FUNCTION_BLOCK TreeStrategyExecutor EXTENDS CNM_AbstractObject.Object IMPLEMENTS CNM_CollectionInterfaces.ITreeStrategy
VAR
	tree :ITreeHelper;
	instantExecutor :InstantTreeStrategyExecutor;
END_VAR

(*

## Short summary

This abstract property returns the class name of the concrete object, 
which is useful for logging/debugging purpose.

.. <legal notes>

legal notes
=================
| SPDX-FileCopyrightText: © 2022 ekvip automation GmbH <info@ekvip.de>
| SPDX-License-Identifier: Apache-2.0
| For details check: Apache-2.0_

.. _Apache-2.0: https://www.apache.org/licenses/LICENSE-2.0

.. </legal notes>

*)
PROPERTY className : CNM_AbstractObject.ClassName
GET
className := 'CNM_Collections.TreeStrategyExecutor';
END_GET
END_PROPERTY

(*

## Short summary

The constructor ``FB_init`` is needed to create an unique hash code.
The hash code is a pseudo random number create with a [xorshift](https://en.wikipedia.org/wiki/Xorshift) algorithm.
It can be overwritten on derivations, because it will be called implicit, ``SUPER^.FB_init()`` is not required.
For more information check: [Behavoir with derived function blocks](https://infosys.beckhoff.com/content/1033/tc3_plc_intro/5482088715.html?id=6983869892358031022).

.. <legal notes>

legal notes
=================
| SPDX-FileCopyrightText: © 2022 ekvip automation GmbH <info@ekvip.de>
| SPDX-License-Identifier: Apache-2.0
| For details check: Apache-2.0_

.. _Apache-2.0: https://www.apache.org/licenses/LICENSE-2.0

.. </legal notes>


*)
METHOD FB_init : BOOL
VAR_INPUT
	(* if TRUE, the retain variables are initialized (warm start / cold start)*)
	bInitRetains	: BOOL;
	(* if TRUE, the instance afterwards gets moved into the copy code (online change) *)
	bInCopyCode	: BOOL;
	(*the tree which this executor will dispatch to*)
	tree :ITreeHelper;
END_VAR
THIS^.tree := tree;
THIS^.instantExecutor.assignTree(tree);
END_METHOD

(*

## Short summary

A method to insert a single element into the tree.

.. <legal notes>

legal notes
=================
| SPDX-FileCopyrightText: © 2022 ekvip automation GmbH <info@ekvip.de>
| SPDX-License-Identifier: Apache-2.0
| For details check: Apache-2.0_

.. _Apache-2.0: https://www.apache.org/licenses/LICENSE-2.0

.. </legal notes>


**Return:** ``SUCCESS``: operation successful
	``ABORTED``: operation was aborted (implementation specific)
	``ERROR``: out of memory

*)
METHOD insert : CNM_CollectionInterfaces.CNM_ReturnTypes.SingleExecutionResult
VAR_INPUT
	(*the object that should be inserted*)
	object	: CNM_CollectionInterfaces.CNM_AbstractObject.IObject;
END_VAR
insert := THIS^.tree.insert(object := object);
END_METHOD

(*

## Short summary

This method inserts all elements of a collection into the tree.

If any value of the collection could not be inserted because of duplication, operation isn't aborted, 
insertion is tried for every element of the collection.

.. <legal notes>

legal notes
=================
| SPDX-FileCopyrightText: © 2025 ekvip automation GmbH <info@ekvip.de>
| SPDX-License-Identifier: Apache-2.0
| For details check: Apache-2.0_

.. _Apache-2.0: https://www.apache.org/licenses/LICENSE-2.0

.. </legal notes>


**Return:** ``SUCCESS``: if insert could be made
	``ABORTED``: execute has a falling edge during insert,
	``BUSY``: Insert is in Progress
	``ERROR``: the passed collection where not valid / contained invalid Elements
	``IDLE``: method was never started

*)
METHOD insertCollection : CNM_CollectionInterfaces.CNM_ReturnTypes.SingleExecutionState
VAR_INPUT
	(*The collection that should be inserted*)
	collection	: CNM_CollectionInterfaces.ICollection;
	(*If insert should be processed*)
	execute	: BOOL;
END_VAR
insertCollection := THIS^.tree.insertCollection(collection := collection, execute := execute);
END_METHOD

(*

## Short summary

This property returns a fluent interface for immediate (wihtin one call) operations of tree.

.. <legal notes>

legal notes
=================
| SPDX-FileCopyrightText: © 2025 ekvip automation GmbH <info@ekvip.de>
| SPDX-License-Identifier: Apache-2.0
| For details check: Apache-2.0_

.. _Apache-2.0: https://www.apache.org/licenses/LICENSE-2.0

.. </legal notes>

*)
PROPERTY instant : CNM_CollectionInterfaces.IInstantTreeStrategy
GET
instant := THIS^.instantExecutor;
END_GET
END_PROPERTY

(*

## Short summary

Function to remove an object from the tree

.. <legal notes>

legal notes
=================
| SPDX-FileCopyrightText: © 2022 ekvip automation GmbH <info@ekvip.de>
| SPDX-License-Identifier: Apache-2.0
| For details check: Apache-2.0_

.. _Apache-2.0: https://www.apache.org/licenses/LICENSE-2.0

.. </legal notes>


**Return:** ``SUCCESS``: if remove could be made
	``ABORTED``: if object wasn't in the tree
	``ERROR``: if object wasn't valid

*)
METHOD remove : CNM_CollectionInterfaces.CNM_ReturnTypes.SingleExecutionResult
VAR_INPUT
	(* The object that should be removed *)
	object	: CNM_CollectionInterfaces.CNM_AbstractObject.IObject;
END_VAR
remove := THIS^.tree.remove(object := object);
END_METHOD

END_FUNCTION_BLOCK

(* stored: Version 1.1.0.1, ProductVersion 3.1.4026.13
   POU TreeStrategyExecutor: Id {f0f69923-1de4-4221-a29f-9b4c582ab374}, SpecialFunc None
   Property className: Id {626201f9-1520-4f11-96e0-880a93fc92e2}
   Get Get: Id {b51ad4c2-946d-4b7d-822f-0ac0d6c0e944}
   Method FB_init: Id {336768f3-f108-411b-9a94-5d6a8f509bb1}
   Method insert: Id {25f6a29e-bb89-4d2a-ab89-b1901021b4bf}
   Method insertCollection: Id {7a4f8576-2e7f-455f-a701-dd1522cb8d25}
   Property instant: Id {1e089ab7-463b-4c55-8d50-6aff869bdd31}
   Get Get: Id {6b2b1536-320e-4be6-abaf-f01b99fa2ecc}
   Method remove: Id {8564183e-f094-440a-a82b-a4691e03216d} *)
